# EPICS substitutions: lsredis/iocBoot/iocCygwin/softMotor.substitutions
file "$(STD)/stdApp/Db/softMotor.db"
{
pattern
{P,		SM}
{lsredis:,	SM1}
{lsredis:,	SM2}
{lsredis:,	SM3}
{lsredis:,	SM4}
{lsredis:,	SM5}
{lsredis:,	SM6}
{lsredis:,	SM7}
{lsredis:,	SM8}
{lsredis:,	SM9}
{lsredis:,	SM10}
}
